FUNCTION_BLOCK Test_WriteBySymbolName_KeepingHandle EXTENDS T_UnitTestBase
VAR
    AdsPort              : UINT;
    AdsWriteBySymbolName : T_AdsWriteBySymbolName;
    AdsReadSymbolName    : T_AdsReadSymbolName;
    WriteResult          : INT; // We are writing to this variable by its symbol name
    State                : INT;
END_VAR

METHOD Init
State := 0;
END_METHOD

{attribute 'analysis' := '-33'} // inhibit unused variable warning
METHOD RunTest
VAR_OUTPUT
    TestCompleted : BOOL;
    TestFailed    : BOOL;
END_VAR
VAR_INST
    SymbolName   : T_MaxString;
    ValueToWrite : INT;
END_VAR
CASE State OF
    0:
        AdsPort      := _AppInfo.AdsPort;
        ValueToWrite := 3456;
        WriteResult  := 0;
        AdsReadSymbolName.Execute(Address := ADR(WriteResult),
                                  Length  := SIZEOF(WriteResult),
                                  PlcPort := AdsPort);
        State := 10;

    10:
        IF NOT AdsReadSymbolName.Execution.Busy THEN
            SymbolName := AdsReadSymbolName.SymbolName;
            State      := 20;
        END_IF

    20:
        AdsWriteBySymbolName.Execute(AmsNetId         := '',
                                     Port             := AdsPort,
                                     SymbolName       := SymbolName,
                                     WriteDataAddress := ADR(ValueToWrite),
                                     WriteDataLength  := SIZEOF(ValueToWrite),
                                     KeepSymbolHandle := TRUE);

        State := 30;

    30:
        IF NOT AdsWriteBySymbolName.Execution.Busy THEN
            State := 40;
        END_IF

    40:
        AssertTrue(Source    := TestName,
                   Condition := (WriteResult = 3456),
                   Message   := 'WriteResult <> 3456',
                   Failed    => TestFailed);

        TestCompleted := TRUE;
END_CASE

AdsWriteBySymbolName();
AdsReadSymbolName();
END_METHOD

END_FUNCTION_BLOCK

(* stored: Version 1.1.0.1, ProductVersion 3.1.4024.12
   POU Test_WriteBySymbolName_KeepingHandle: Id {cbd57208-6859-0aad-17cb-ff3a12b998ac}, SpecialFunc None
   Method Init: Id {c428c6fe-957d-06a0-2d47-21b92364bc9c}
   Method RunTest: Id {c4f343de-bf0c-04fa-343e-61fca8cd8dfe} *)
